// TIA Portal V20 export
DATA_BLOCK "SBK5"   // DB289
// stored: MemoryReserve 100
   VAR
      "X1-1 SCS BOX SCS MODE SLELECT SS.SETUP" : Bool;
      "X2-1 SCS BOX SCS MODE SLELECT SS.DISABLE" : Bool;
      "X3-1 SPARE" : Bool;
      "X4-1 SPARE" : Bool;
      "X1-2 SCS BOX SCS MODE SLELECT SS.AUTO" : Bool;
      "X2-2 SPARE" : Bool;
      "X3-2 SPARE" : Bool;
      "X4-2 SPARE" : Bool;
   END_VAR
BEGIN
END_DATA_BLOCK
